FUNCTION_BLOCK IOHandler (* Composite Function Block Type *)
  (* Standard: 61499-2 *)
  (* Version 0.0, 9/6/2016, Dmitry, nxtControl GmbH, template *)
  PACKAGE Main;
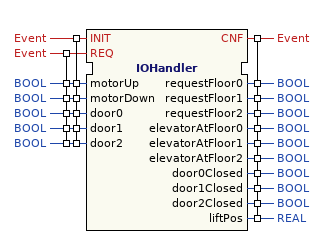
  EVENT_INPUT
    INIT WITH motorUp, motorDown, door0, door1, door2; (* Initialization Request *)
    REQ WITH motorUp, motorDown, door0, door1, door2; (* Normal Execution Request *)
  END_EVENT
  EVENT_OUTPUT
    CNF WITH requestFloor0, requestFloor1, requestFloor2, elevatorAtFloor0, elevatorAtFloor1, elevatorAtFloor2, door0Closed, door1Closed, door2Closed, liftPos; (* Execution Confirmation *)
  END_EVENT
  VAR_INPUT
    motorUp : BOOL; (* Input event qualifier *)
    motorDown : BOOL;
    door0 : BOOL;
    door1 : BOOL;
    door2 : BOOL;
  END_VAR
  VAR_OUTPUT
    requestFloor0 : BOOL;
    requestFloor1 : BOOL;
    requestFloor2 : BOOL;
    elevatorAtFloor0 : BOOL;
    elevatorAtFloor1 : BOOL;
    elevatorAtFloor2 : BOOL;
    door0Closed : BOOL;
    door1Closed : BOOL;
    door2Closed : BOOL;
    liftPos : REAL;
  END_VAR
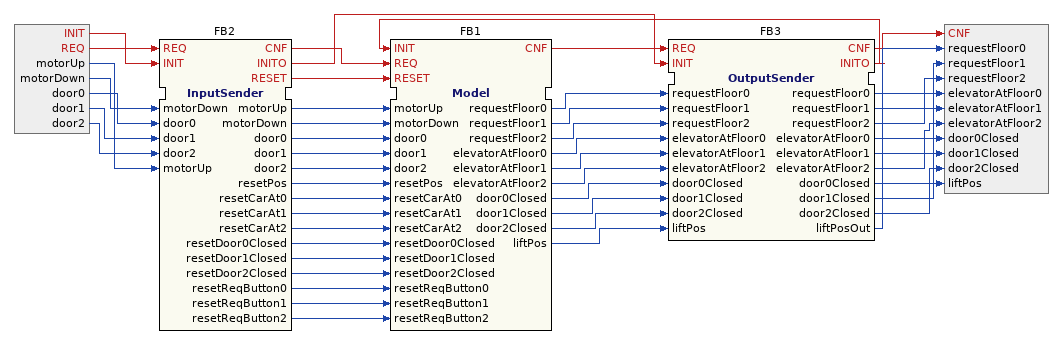
  FBS
    FB2 : InputSender;
    FB1 : Model;
    FB3 : OutputSender;
  END_FBS
  EVENT_CONNECTIONS
    REQ TO FB2.REQ;
    FB1.CNF TO FB3.REQ;
    FB3.CNF TO CNF;
    INIT TO FB2.INIT;
    FB3.INITO TO FB1.INIT;
    FB2.CNF TO FB1.REQ;
    FB2.INITO TO FB3.INIT;
    FB2.RESET TO FB1.RESET;
  END_CONNECTIONS
  DATA_CONNECTIONS
    motorDown TO FB2.motorDown;
    door0 TO FB2.door0;
    door1 TO FB2.door1;
    door2 TO FB2.door2;
    motorUp TO FB2.motorUp;
    FB1.requestFloor0 TO FB3.requestFloor0;
    FB1.requestFloor1 TO FB3.requestFloor1;
    FB1.requestFloor2 TO FB3.requestFloor2;
    FB1.elevatorAtFloor0 TO FB3.elevatorAtFloor0;
    FB1.elevatorAtFloor1 TO FB3.elevatorAtFloor1;
    FB1.elevatorAtFloor2 TO FB3.elevatorAtFloor2;
    FB1.door0Closed TO FB3.door0Closed;
    FB1.door1Closed TO FB3.door1Closed;
    FB1.door2Closed TO FB3.door2Closed;
    FB1.liftPos TO FB3.liftPos;
    FB3.requestFloor0 TO requestFloor0;
    FB3.requestFloor1 TO requestFloor1;
    FB3.requestFloor2 TO requestFloor2;
    FB3.elevatorAtFloor0 TO elevatorAtFloor0;
    FB3.elevatorAtFloor1 TO elevatorAtFloor1;
    FB3.elevatorAtFloor2 TO elevatorAtFloor2;
    FB3.door0Closed TO door0Closed;
    FB3.door1Closed TO door1Closed;
    FB3.door2Closed TO door2Closed;
    FB2.motorUp TO FB1.motorUp;
    FB2.motorDown TO FB1.motorDown;
    FB2.door0 TO FB1.door0;
    FB2.door1 TO FB1.door1;
    FB2.door2 TO FB1.door2;
    FB3.liftPosOut TO liftPos;
    FB2.resetPos TO FB1.resetPos;
    FB2.resetCarAt0 TO FB1.resetCarAt0;
    FB2.resetCarAt1 TO FB1.resetCarAt1;
    FB2.resetCarAt2 TO FB1.resetCarAt2;
    FB2.resetDoor0Closed TO FB1.resetDoor0Closed;
    FB2.resetDoor1Closed TO FB1.resetDoor1Closed;
    FB2.resetDoor2Closed TO FB1.resetDoor2Closed;
    FB2.resetReqButton0 TO FB1.resetReqButton0;
    FB2.resetReqButton1 TO FB1.resetReqButton1;
    FB2.resetReqButton2 TO FB1.resetReqButton2;
  END_CONNECTIONS
END_FUNCTION_BLOCK
